Fanuc KAREL source: kt00533.KL

-- PROVISIONAL review KL for V1013-1; original PC SHA256 7972114a0231bab8854e52d434c268985a33028c4d0e64e18669c74acb64d2f4
-- Incomplete behavior may be omitted. Consult companion uncertainty JSON. Do not deploy.
PROGRAM KT00533
%NOLOCKGROUP
VAR
  OUT : BOOLEAN
-- UNRESOLVED_DECL P1 type=000199
-- UNRESOLVED_DECL P2 type=000101
BEGIN
  -- UNRESOLVED_PC offsets 5-33; opcodes 49,7E,49,AC,23
  -- UNRESOLVED_PC offsets 38-42; opcodes 7F
END KT00533
